// TIA Portal V17 export
// export: Created 2025-06-25T13:13:21.8538789Z, ExportSetting WithDefaults, DisplayName Totally Integrated Automation Portal, DisplayVersion V17 Update 8, DisplayName TIA Portal Openness, DisplayVersion V17 Update 8, DisplayName TIA Portal Version Control Interface, DisplayVersion V17, DisplayName STEP 7 Professional, DisplayVersion V17 Update 8, DisplayName STEP 7 Safety, DisplayVersion V17 Update 6, DisplayName WinCC Advanced, DisplayVersion V17 Update 8
FUNCTION_BLOCK "fbPIP_Regulator"   // FB28, FBD
TITLE = Position-velocity regulator (PI-P form)
{ S7_Optimized_Access := 'TRUE' }
AUTHOR : Heaten
VERSION : 0.1
// stored: AutoNumber true, IsIECCheckEnabled false, IsRetainMemResEnabled false, MemoryReserve 0, SetENOAutomatically false, UDAEnableTagReadback false
   VAR_INPUT
      sPV : "stCalcValue";   // Process value (position)
      sPVvel : "stCalcValue";   // Process value (velocity)
      fFeedback : Real;   // Output feedback (eg valve %, motor rpm)
      fCycleTime : Real;
      bEnable : Bool;
      bReset : Bool;
   END_VAR
   VAR_OUTPUT
      fOut : Real;
      bAtMin : Bool;
      bAtMax : Bool;
   END_VAR
   VAR_IN_OUT
      sTag : "stPIP_Regulator";
   END_VAR
   VAR
      Outer : Struct   // Outer loop = PI control
         D_Mem : Real;
         I_Mem : Real;
         Param_Mem : Real;
      END_STRUCT;
      Inner : Struct   // Inner loop = P control
         D_Mem : Real;
         I_Mem : Real;
         Param_Mem : Real;
      END_STRUCT;
      fSPVel : Real;
   END_VAR
   VAR_TEMP
      Enabled : Bool;
      fDeviation : Real;
      fDeviationVel : Real;
      bPI_AtMax : Bool;
      bPI_AtMin : Bool;
   END_VAR
BEGIN

REGION Network 1 (SCL): Comments and history
   // Position-velocity controller, cascaded PI-P form
   // 
   //                ___   pos   ____   vel   ___   vel   ___   out   __________         ______
   // pos ref ----> | Σ | ----> | PI | ----> | Σ | ----> | P | ----> | Actuator | ----> | Load |
   //             + |___| error |____|  ref  |___| error |___|       |__________|       |______|
   //                 ^ -                      ^ -                    _______               | 
   //                 |                        |_____________________| dP/dt |______________| measured velocity
   //                 |                                              |_______|              |
   //                 |_____________________________________________________________________| measured position
   //                 
   // For example, heating up a heat exchanger to a certain temperature without exceeding the temperature rise limit
   // 
   // Tuning Steps
   //
   // 1. Set the P constants of both controllers equal to 0, and integral to 9999. By default, the integral limit of the velocity
   //    controller should be set to the actuator's maximum position (eg 100%), and the integral limit of position
   //    controller should be set to the process max velocity (eg 5K/min).
   //
   // Important:from this step forth, the step response of position controller should always be evaluated.
   //
   // 2. Tune the KpVel parameter of the velocity controller. Increase the Kp of both position and velocity 
   //    controllers with a ratio of 10 (Kp_velocity = 10 * Kp_position). Once the real position starts to follow the
   //    reference position, stop increasing the Kp_position and only focus on increasing the Kp_velocity. Increase
   //    (sharpen) the velocity controller as much as possible. As a rule of thumb, increase kP_velocity until you get
   //    close to the instability margin (at this margin, you will feel a vibration effect and some acoustic noise
   //    which is because of controller sharpness). Now, you can reduce kP_velocity to 90% of its value to increase 
   //    the stability margin, and remove vibration noise.
   // 
   // 3. Now that the velocity controller is tuned, it is time to tune the parameters of the PID position 
   //    controller. Start with kP_position, and increase it until you again get close to the instability margin, and 
   //    then reduce kP_position to its 90%. So far, the proportional parts of both inner velocity loop and outer 
   //    position loop are tuned.
   //
   // 4. In this step, increase kI to eliminate the steady state error. As a suggestion start with kI equal to
   //    0.01, and in each step, increase it with a factor of 2. Increase kI step by step until the following two 
   //    conditions are met at the same time: - the overshoot is in its acceptable range - the steady-state error is 
   //    eliminated in a short enough period of time.
END_REGION

REGION Network 3: Reset manual mode
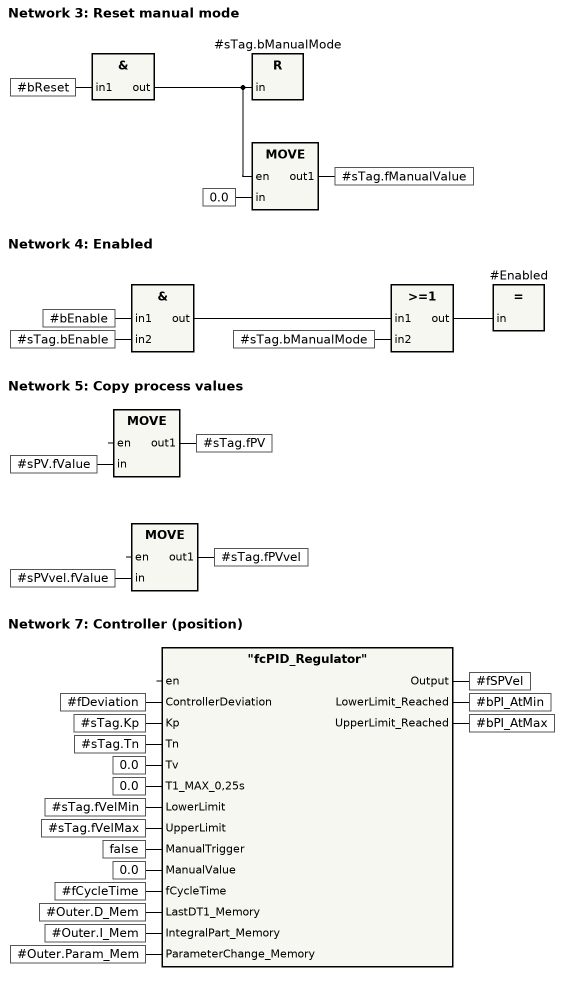
   IF #bReset THEN
       #sTag.bManualMode := FALSE;
       #sTag.fManualValue := 0.0;
   END_IF;
END_REGION

REGION Network 4: Enabled
   // Local input is from process control logic: when to run the regulator
   // Tag input is from HMI: do we want to run this regulator at all
   #Enabled := (#bEnable AND #sTag.bEnable) OR #sTag.bManualMode;
END_REGION

REGION Network 5: Copy process values
   #sTag.fPV := #sPV.fValue;
   #sTag.fPVvel := #sPVvel.fValue;
END_REGION

REGION Network 6 (SCL): Deviation (position)
   // NaN detection
   IF "isNaN"(#sTag.fSP) OR "isNaN"(#sTag.fPV) THEN
       #fDeviation := 0.0;
       #sTag.bFault := TRUE;
   ELSE
       #fDeviation := #sTag.fSP - #sTag.fPV;
       #sTag.bFault := FALSE;
   END_IF;
END_REGION

REGION Network 7: Controller (position)
   // NOTE: controller always runs regardless of mode.
   // This stage generates a velocity setpoint from the position error.
   // Max & min limits are of VELOCITY, this is not abug.
   "fcPID_Regulator"(ControllerDeviation := #fDeviation,
                     Kp := #sTag.Kp,
                     Tn := #sTag.Tn,
                     Tv := 0.0,
                     "T1_MAX_0,25s" := 0.0,
                     LowerLimit := #sTag.fVelMin,
                     UpperLimit := #sTag.fVelMax,
                     ManualTrigger := false,
                     ManualValue := 0.0,
                     fCycleTime := #fCycleTime,
                     LastDT1_Memory := #Outer.D_Mem,
                     IntegralPart_Memory := #Outer.I_Mem,
                     ParameterChange_Memory := #Outer.Param_Mem,
                     Output => #fSPVel,
                     LowerLimit_Reached => #bPI_AtMin,
                     UpperLimit_Reached => #bPI_AtMax);
END_REGION

REGION Network 8 (SCL): Deviation (velocity)
   // NaN detection
   IF "isNaN"(#sTag.fPVvel) THEN
       #fDeviationVel := 0.0;
       #sTag.bFault := TRUE;
   ELSE
       #fDeviationVel := #fSPVel - #sTag.fPVvel;
       #sTag.bFault := FALSE;
   END_IF;
END_REGION

REGION Network 9: Controller (velocity)
   // NOTE: controller always runs regardless of mode
   // This stage generates the manipulated value from the velocity error.
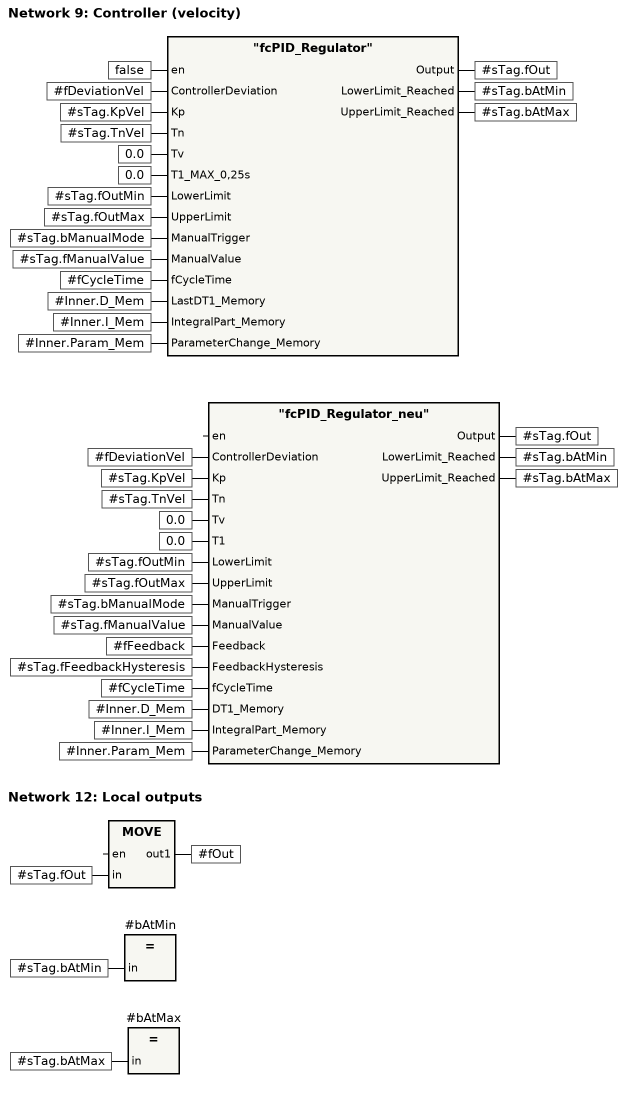
   IF false THEN
       "fcPID_Regulator"(ControllerDeviation := #fDeviationVel,
                         Kp := #sTag.KpVel,
                         Tn := #sTag.TnVel,
                         Tv := 0.0,
                         "T1_MAX_0,25s" := 0.0,
                         LowerLimit := #sTag.fOutMin,
                         UpperLimit := #sTag.fOutMax,
                         ManualTrigger := #sTag.bManualMode,
                         ManualValue := #sTag.fManualValue,
                         fCycleTime := #fCycleTime,
                         LastDT1_Memory := #Inner.D_Mem,
                         IntegralPart_Memory := #Inner.I_Mem,
                         ParameterChange_Memory := #Inner.Param_Mem,
                         Output => #sTag.fOut,
                         LowerLimit_Reached => #sTag.bAtMin,
                         UpperLimit_Reached => #sTag.bAtMax);
   END_IF;
   "fcPID_Regulator_neu"(ControllerDeviation := #fDeviationVel,
                         Kp := #sTag.KpVel,
                         Tn := #sTag.TnVel,
                         Tv := 0.0,
                         T1 := 0.0,
                         LowerLimit := #sTag.fOutMin,
                         UpperLimit := #sTag.fOutMax,
                         ManualTrigger := #sTag.bManualMode,
                         ManualValue := #sTag.fManualValue,
                         Feedback := #fFeedback,
                         FeedbackHysteresis := #sTag.fFeedbackHysteresis,
                         fCycleTime := #fCycleTime,
                         DT1_Memory := #Inner.D_Mem,
                         IntegralPart_Memory := #Inner.I_Mem,
                         ParameterChange_Memory := #Inner.Param_Mem,
                         Output => #sTag.fOut,
                         LowerLimit_Reached => #sTag.bAtMin,
                         UpperLimit_Reached => #sTag.bAtMax);
END_REGION

REGION Network 10 (SCL): Disable
   IF #Enabled = FALSE OR #sTag.bFault = TRUE THEN
       #sTag.fOut := 0.0;
       #sTag.bAtMin := FALSE;
       #sTag.bAtMax := FALSE;
   END_IF;
END_REGION

REGION Network 11 (SCL): Mode
   // Mode
   IF #sTag.bManualMode = TRUE THEN
       #sTag.nMode := 2;
   ELSIF #sTag.bEnable = TRUE THEN
       #sTag.nMode := 1;
   ELSE
       #sTag.nMode := 0;
   END_IF;
END_REGION

REGION Network 12: Local outputs
   #fOut := #sTag.fOut;
   #bAtMin := #sTag.bAtMin;
   #bAtMax := #sTag.bAtMax;
END_REGION
END_FUNCTION_BLOCK
